PROGRAM MAIN
VAR
END_VAR

END_PROGRAM

(* stored: Version 1.1.0.1
   POU MAIN: Id {f94b5d02-9944-4b96-a5c8-57cfccdc367f} *)
